FUNCTION_BLOCK MUL_4 (* Calculate arithmetical product of numeric inputs (generic FB) *)
  (* Standard: 61131-3; Classification: standard arithmetic function; Description: Copyright (c) 2026 HR Agrartechnik GmbH This program and the accompanying materials are made available under the terms of the Eclipse Public License 2.0 which is available at https://www.eclipse.org/legal/epl-2.0/ SPDX-License-Identifier: EPL-2.0 *)
  (* Version 1.0, 2026-08-28, Franz Höpfinger, HR Agrartechnik GmbH, initial API and implementation and/or initial documentation *)
  PACKAGE iec61131::arithmetic;
  {SET_ATTRIBUTE(eclipse4diac::core::GenericClassName, 'GEN_MUL')}
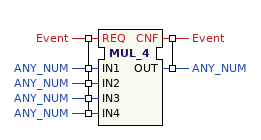
  EVENT_INPUT
    REQ WITH IN1, IN2, IN3, IN4; (* Normal Execution Request *)
  END_EVENT
  EVENT_OUTPUT
    CNF WITH OUT; (* Execution Confirmation *)
  END_EVENT
  VAR_INPUT
    IN1 : ANY_NUM; (* MUL input 1 *)
    IN2 : ANY_NUM; (* MUL input 2 *)
    IN3 : ANY_NUM; (* MUL input 3 *)
    IN4 : ANY_NUM; (* MUL input 4 *)
  END_VAR
  VAR_OUTPUT
    OUT : ANY_NUM; (* MUL result *)
  END_VAR
END_FUNCTION_BLOCK
